// TIA Portal V20 export
FUNCTION "EM13_TeachingData" : Void   // FC87, LAD
// stored: Namespace Unit1.Em13, SetENOAutomatically false
BEGIN

REGION Network 2 (SCL): JR Unloading PnP AxisX Teaching Position
   // Transfer PnP Left AxisX Position 0
   "Unit1.Em13.HmiInterface".cmJRUnloadingPnPAxisX.configuration.setPositions[0].position := 1265.0;
   "Unit1.Em13.HmiInterface".cmJRUnloadingPnPAxisX.configuration.setPositions[0].velocity := 50.0;

   // Transfer PnP Left AxisX Position 1
   "Unit1.Em13.HmiInterface".cmJRUnloadingPnPAxisX.configuration.setPositions[1].position := 873.5;
   "Unit1.Em13.HmiInterface".cmJRUnloadingPnPAxisX.configuration.setPositions[1].velocity := 50.0;

   // Transfer PnP Left AxisX Position 2
   "Unit1.Em13.HmiInterface".cmJRUnloadingPnPAxisX.configuration.setPositions[2].position := 480.0;
   "Unit1.Em13.HmiInterface".cmJRUnloadingPnPAxisX.configuration.setPositions[2].velocity := 50.0;

   // Transfer PnP Left AxisX Position 3
   "Unit1.Em13.HmiInterface".cmJRUnloadingPnPAxisX.configuration.setPositions[3].position := 1265.0;
   "Unit1.Em13.HmiInterface".cmJRUnloadingPnPAxisX.configuration.setPositions[3].velocity := 50.0;

   // Transfer PnP Left AxisX Position 4
   "Unit1.Em13.HmiInterface".cmJRUnloadingPnPAxisX.configuration.setPositions[4].position := 1265.0;
   "Unit1.Em13.HmiInterface".cmJRUnloadingPnPAxisX.configuration.setPositions[4].velocity := 50.0;

   // Transfer PnP Left AxisX Position 5
   "Unit1.Em13.HmiInterface".cmJRUnloadingPnPAxisX.configuration.setPositions[5].position := 26.47;
   "Unit1.Em13.HmiInterface".cmJRUnloadingPnPAxisX.configuration.setPositions[5].velocity := 50.0;

   //////////////////////// ZONE ///////////////////////
   "Unit1.Em13.HmiInterface".cmJRUnloadingPnPAxisX.configuration.setPositions[9].position := 107.84;
   "Unit1.Em13.HmiInterface".cmJRUnloadingPnPAxisX.configuration.setPositions[9].velocity := 50.0;

   "Unit1.Em13.HmiInterface".cmJRUnloadingPnPAxisX.configuration.setPositions[10].position := 1300.0;
   "Unit1.Em13.HmiInterface".cmJRUnloadingPnPAxisX.configuration.setPositions[10].velocity := 50.0;
END_REGION

REGION Network 3 (SCL): JR Unloading PnP AxisC Teaching Position
   // Transfer PnP Left AxisY Position 0
   "Unit1.Em13.HmiInterface".cmJRUnloadingPnPAxisC.configuration.setPositions[0].position := -88.0;
   "Unit1.Em13.HmiInterface".cmJRUnloadingPnPAxisC.configuration.setPositions[0].velocity := 10.0;

   // Transfer PnP Left AxisY Position 1
   "Unit1.Em13.HmiInterface".cmJRUnloadingPnPAxisC.configuration.setPositions[1].position := 178.0;
   "Unit1.Em13.HmiInterface".cmJRUnloadingPnPAxisC.configuration.setPositions[1].velocity := 10.0;

   // Transfer PnP Left AxisY Position 2
   "Unit1.Em13.HmiInterface".cmJRUnloadingPnPAxisC.configuration.setPositions[2].position := -88.0;
   "Unit1.Em13.HmiInterface".cmJRUnloadingPnPAxisC.configuration.setPositions[2].velocity := 10.0;

   // Transfer PnP Left AxisY Position 3
   "Unit1.Em13.HmiInterface".cmJRUnloadingPnPAxisC.configuration.setPositions[3].position := -88.0;
   "Unit1.Em13.HmiInterface".cmJRUnloadingPnPAxisC.configuration.setPositions[3].velocity := 10.0;

   // Transfer PnP Left AxisY Position 4
   "Unit1.Em13.HmiInterface".cmJRUnloadingPnPAxisC.configuration.setPositions[4].position := 178.0;
   "Unit1.Em13.HmiInterface".cmJRUnloadingPnPAxisC.configuration.setPositions[4].velocity := 10.0;

   //////////////////////// ZONE ///////////////////////
   "Unit1.Em13.HmiInterface".cmJRUnloadingPnPAxisC.configuration.setPositions[10].position := -90.0;
   "Unit1.Em13.HmiInterface".cmJRUnloadingPnPAxisC.configuration.setPositions[10].velocity := 10.0;
END_REGION

REGION Network 4 (SCL): JR Unloading PnP AxisZ Teaching Position
   // Transfer PnP Left AxisZ Position 0
   "Unit1.Em13.HmiInterface".cmJRUnloadingPnPAxisZ.configuration.setPositions[0].position := 0.0;
   "Unit1.Em13.HmiInterface".cmJRUnloadingPnPAxisZ.configuration.setPositions[0].velocity := 10.0;

   // Transfer PnP Left AxisZ Position 1
   "Unit1.Em13.HmiInterface".cmJRUnloadingPnPAxisZ.configuration.setPositions[1].position := 211.0;
   "Unit1.Em13.HmiInterface".cmJRUnloadingPnPAxisZ.configuration.setPositions[1].velocity := 10.0;

   // Transfer PnP Left AxisZ Position 2
   "Unit1.Em13.HmiInterface".cmJRUnloadingPnPAxisZ.configuration.setPositions[2].position := 0.0;
   "Unit1.Em13.HmiInterface".cmJRUnloadingPnPAxisZ.configuration.setPositions[2].velocity := 10.0;

   // Transfer PnP Left AxisZ Position 3
   "Unit1.Em13.HmiInterface".cmJRUnloadingPnPAxisZ.configuration.setPositions[3].position := 0.0;
   "Unit1.Em13.HmiInterface".cmJRUnloadingPnPAxisZ.configuration.setPositions[3].velocity := 10.0;

   // Transfer PnP Left AxisZ Position 4
   "Unit1.Em13.HmiInterface".cmJRUnloadingPnPAxisZ.configuration.setPositions[4].position := 157.5;
   "Unit1.Em13.HmiInterface".cmJRUnloadingPnPAxisZ.configuration.setPositions[4].velocity := 10.0;


   //////////////////////// ZONE ///////////////////////
   "Unit1.Em13.HmiInterface".cmJRUnloadingPnPAxisX.configuration.setPositions[9].position := 0;
   "Unit1.Em13.HmiInterface".cmJRUnloadingPnPAxisX.configuration.setPositions[9].velocity := 0.0;
END_REGION
END_FUNCTION
